// TIA Portal V19 export
FUNCTION_BLOCK "GuideLubrication_FB"   // FB155, LAD
TITLE = GUIDE LUBRICATION / MATERIAL LUBRICATION (ROLL)
// stored: Access Published, MemoryReserve 100, SetENOAutomatically false
   VAR_INPUT
      AreaInterface : "AreaInterface";
      DataIn : Struct
         PbCycleExe : Bool;
         FluxCycleDone : Bool;
         SensorLevel : Bool;
         PumpFeedbackRunning : Bool;
         PumpThermalProtection : Bool;
      END_STRUCT;
      CIn : Struct
         EnableStopInPhase : Bool;
         EnableStopProgrammed : Bool;
         MaterialCounter : LReal;
      END_STRUCT;
      Config : Struct
         EnableWngSystemOff : Bool;
         LowTankLevelDly : Time;
      END_STRUCT;
   END_VAR
   VAR_OUTPUT
      MachineInterface : "MachineInterface";
      DataOut : Struct
         M_Pump_Contactor : Bool;
         Lamp : Bool;
      END_STRUCT;
      COut : Struct
         PumpIsRunning : Bool;
      END_STRUCT;
   END_VAR
   VAR_IN_OUT
      PersistentValues : Struct
         Par : Struct
            Enable : Bool;
            CycleToExecute : Int;
            SpaceInterval : LReal;
         END_STRUCT;
      END_STRUCT;
   END_VAR
   VAR
      Sts : Struct
         AlarmsPresence : Bool;
         WarningsPresence : Bool;
         IsStandstill : Bool;
         PumpRunReq : Bool;
         LastFeed : LReal;
         PrevMatcounter : LReal;
         MaterialFed : LReal;
         PumpCnd { ExternalAccessible := 'False'; ExternalVisible := 'False'; ExternalWritable := 'False'} : Bool;
         CycleDone : Int;
      END_STRUCT;
      Ctrl : Struct
         RstAlarms : Bool;
         StopInPhase : Bool;
         StopProgrammed : Bool;
         PumpStart : Bool;
      END_STRUCT;
      Alr : Struct
         LowTankLevel : Bool;
         TimeoutCycle : Bool;
         MPump : "MotorAlr";
      END_STRUCT;
      Wng : Struct
         NoAutReady : Bool;
         SystemOff : Bool;
      END_STRUCT;
      M_Pump : "Motor";
      TON_DelayBlowerStop { S7_SetPoint := 'True'} : IEC_TIMER;
      TON_DelayPumpStop { S7_SetPoint := 'True'} : IEC_TIMER;
      TON_LowTankLevel { S7_SetPoint := 'True'} : IEC_TIMER;
      TON_CycleTimeout { S7_SetPoint := 'True'} : IEC_TIMER;
      AckRstAlarms : Bool;
      PbCycleStart_PEAux : Bool;
      CycleDone_PEAux : Bool;
   END_VAR
   VAR_TEMP
      CycleDone_PE : Bool;
   END_VAR
   VAR_TEMP   // added for the SCL form of the ladder/FBD networks
      _w1 : Bool;
   END_VAR
BEGIN

REGION Network 1 (SCL): Reset alarms command
   #Ctrl.RstAlarms := #AreaInterface.RstAlarms AND NOT #AckRstAlarms; 
   #AckRstAlarms := #AreaInterface.RstAlarms;

   IF #Ctrl.RstAlarms THEN
       #Wng.NoAutReady := FALSE;
       #Alr.LowTankLevel := FALSE;
       #Alr.TimeoutCycle := FALSE;
   END_IF;
END_REGION

REGION Network 2: Warning Pump off / Warning Pump / Blower off
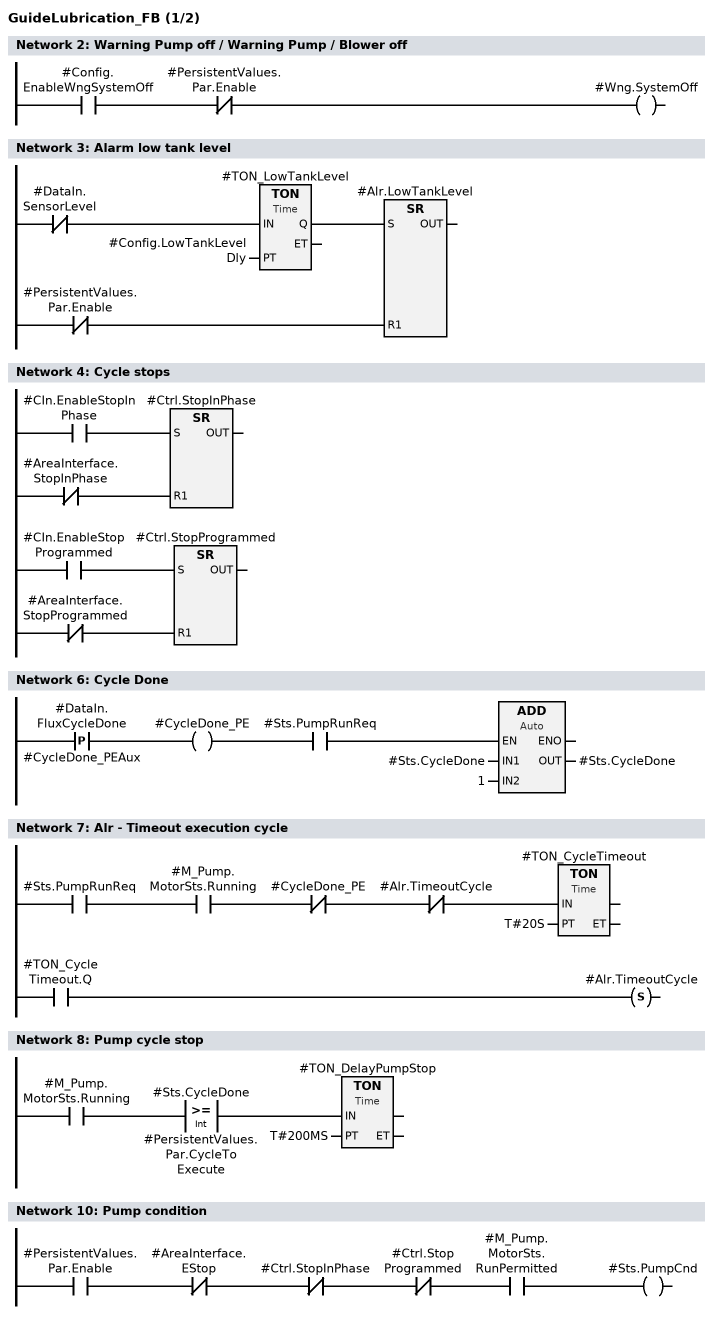
   RUNG wire#powerrail
      Contact( #Config.EnableWngSystemOff )
      I_Contact( #PersistentValues.Par.Enable )
      Coil( #Wng.SystemOff )
   END_RUNG
   // the same network as SCL:
   #Wng.SystemOff := #Config.EnableWngSystemOff AND NOT #PersistentValues.Par.Enable;
END_REGION

REGION Network 3: Alarm low tank level
   RUNG wire#powerrail
      I_Contact( #DataIn.SensorLevel )
      { S7_Templates := "time_type := Time" } #TON_LowTankLevel.TON(pt := #Config.LowTankLevelDly, et =>)
      S_SR(operand := #Alr.LowTankLevel, r1 := wire#w1)
   END_RUNG
   RUNG wire#powerrail
      I_Contact( #PersistentValues.Par.Enable )
   END_RUNG wire#w1
   // the same network as SCL:
   #TON_LowTankLevel.TON(IN := NOT #DataIn.SensorLevel, PT := #Config.LowTankLevelDly);
   IF #TON_LowTankLevel.Q THEN
       #Alr.LowTankLevel := TRUE;   // SR flip-flop
   END_IF;
   IF NOT #PersistentValues.Par.Enable THEN #Alr.LowTankLevel := FALSE; END_IF;
END_REGION

REGION Network 4: Cycle stops
   RUNG wire#powerrail
      Contact( #CIn.EnableStopInPhase )
      S_SR(operand := #Ctrl.StopInPhase, r1 := wire#w1)
   END_RUNG
   RUNG wire#powerrail
      I_Contact( #AreaInterface.StopInPhase )
   END_RUNG wire#w1
   RUNG wire#powerrail
      Contact( #CIn.EnableStopProgrammed )
      S_SR(operand := #Ctrl.StopProgrammed, r1 := wire#w2)
   END_RUNG
   RUNG wire#powerrail
      I_Contact( #AreaInterface.StopProgrammed )
   END_RUNG wire#w2
   // the same network as SCL:
   IF #CIn.EnableStopInPhase THEN
       #Ctrl.StopInPhase := TRUE;   // SR flip-flop
   END_IF;
   IF NOT #AreaInterface.StopInPhase THEN #Ctrl.StopInPhase := FALSE; END_IF;
   IF #CIn.EnableStopProgrammed THEN
       #Ctrl.StopProgrammed := TRUE;   // SR flip-flop
   END_IF;
   IF NOT #AreaInterface.StopProgrammed THEN #Ctrl.StopProgrammed := FALSE; END_IF;
END_REGION

REGION Network 5: <<< PUMP >>>
END_REGION

REGION Network 6: Cycle Done
   RUNG wire#powerrail
      P_Contact(operand := #DataIn.FluxCycleDone, bit := #CycleDone_PEAux)
      Coil( #CycleDone_PE )
      Contact( #Sts.PumpRunReq )
      Add(in1 := #Sts.CycleDone, in2 := 1, out => #Sts.CycleDone)
   END_RUNG
   // the same network as SCL:
   #_w1 := #DataIn.FluxCycleDone AND NOT #CycleDone_PEAux;   // rising edge of #DataIn.FluxCycleDone
   #CycleDone_PEAux := #DataIn.FluxCycleDone;
   #CycleDone_PE := #_w1;
   IF #_w1 AND #Sts.PumpRunReq THEN #Sts.CycleDone := #Sts.CycleDone + 1; END_IF;
END_REGION

REGION Network 7: Alr - Timeout execution cycle
   RUNG wire#powerrail
      Contact( #Sts.PumpRunReq )
      Contact( #M_Pump.MotorSts.Running )
      I_Contact( #CycleDone_PE )
      I_Contact( #Alr.TimeoutCycle )
      { S7_Templates := "time_type := Time" } #TON_CycleTimeout.TON(pt := T#20S, et =>)
   END_RUNG
   RUNG wire#powerrail
      Contact( #TON_CycleTimeout.Q )
      S_Coil( #Alr.TimeoutCycle )
   END_RUNG
   // the same network as SCL:
   #TON_CycleTimeout.TON(IN := #Sts.PumpRunReq AND #M_Pump.MotorSts.Running AND NOT #CycleDone_PE AND NOT #Alr.TimeoutCycle,
                         PT := T#20S);
   IF #TON_CycleTimeout.Q THEN #Alr.TimeoutCycle := TRUE; END_IF;
END_REGION

REGION Network 8: Pump cycle stop
   RUNG wire#powerrail
      Contact( #M_Pump.MotorSts.Running )
      { S7_Templates := "SrcType := Int" } GE_Contact(in1 := #Sts.CycleDone, in2 := #PersistentValues.Par.CycleToExecute)
      { S7_Templates := "time_type := Time" } #TON_DelayPumpStop.TON(pt := T#200MS, et =>)
   END_RUNG
   // the same network as SCL:
   #TON_DelayPumpStop.TON(IN := #M_Pump.MotorSts.Running AND (#Sts.CycleDone >= #PersistentValues.Par.CycleToExecute),
                          PT := T#200MS);
END_REGION

REGION Network 9 (SCL): Pump run request
   #Sts.LastFeed := "M_PosAMinusPosB"(PosA:=#CIn.MaterialCounter,PosB:=#Sts.PrevMatcounter,MODULE := "MATERIAL_COUNTERS_MODULE");
   #Sts.PrevMatcounter := #CIn.MaterialCounter;

   IF #Sts.LastFeed > 1000.0 THEN
       #Sts.LastFeed := 0;
   END_IF;

   #Sts.MaterialFed := #Sts.MaterialFed + #Sts.LastFeed;

   IF  #PersistentValues.Par.CycleToExecute = 0 OR #PersistentValues.Par.SpaceInterval <= 0.0 OR NOT #PersistentValues.Par.Enable THEN
       #Sts.PumpRunReq := FALSE;       
   ELSIF #TON_DelayPumpStop.Q THEN
       #Sts.PumpRunReq := FALSE;   
       #Sts.MaterialFed := 0.0;
       #Sts.CycleDone := 0;
   ELSIF NOT #Sts.PumpRunReq AND (#Sts.MaterialFed >= #PersistentValues.Par.SpaceInterval OR #DataIn.PbCycleExe) THEN
       #Sts.PumpRunReq := TRUE;
       #Sts.CycleDone := 0;
   END_IF;
END_REGION

REGION Network 10: Pump condition
   RUNG wire#powerrail
      Contact( #PersistentValues.Par.Enable )
      I_Contact( #AreaInterface.EStop )
      I_Contact( #Ctrl.StopInPhase )
      I_Contact( #Ctrl.StopProgrammed )
      Contact( #M_Pump.MotorSts.RunPermitted )
      Coil( #Sts.PumpCnd )
   END_RUNG
   // the same network as SCL:
   #Sts.PumpCnd := #PersistentValues.Par.Enable AND NOT #AreaInterface.EStop AND NOT #Ctrl.StopInPhase AND NOT #Ctrl.StopProgrammed AND #M_Pump.MotorSts.RunPermitted;
END_REGION

REGION Network 11: Pump automatic start
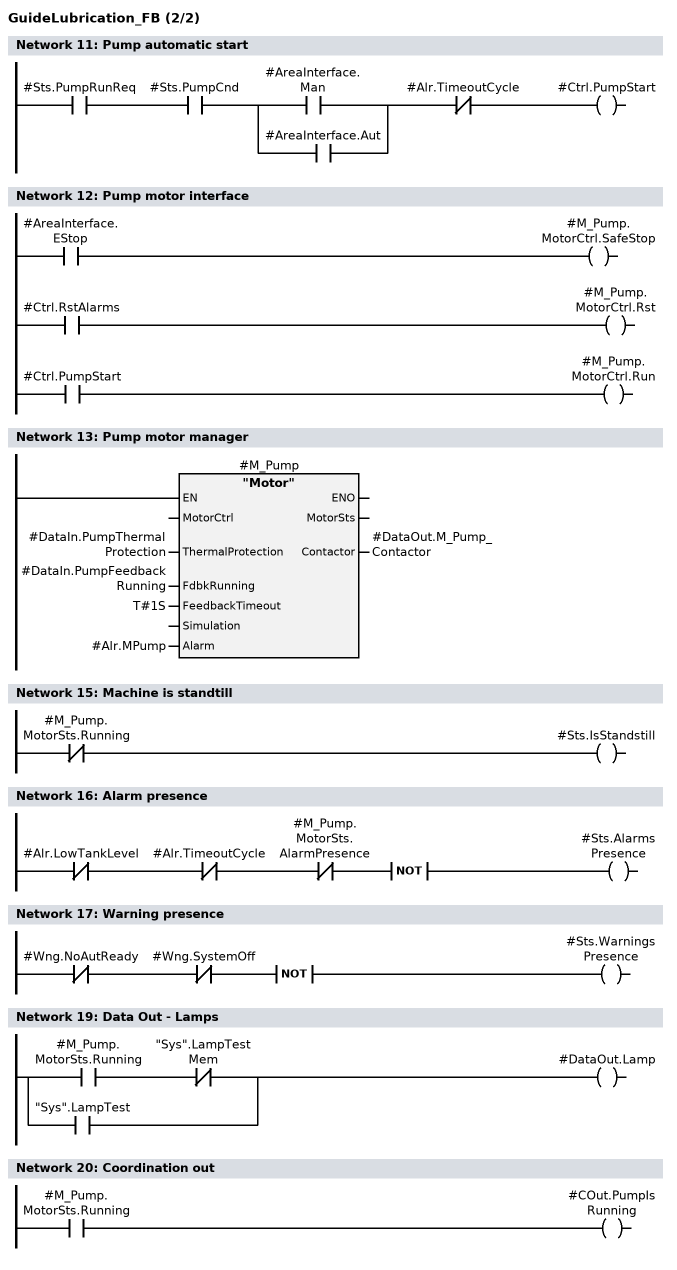
   RUNG wire#powerrail
      Contact( #Sts.PumpRunReq )
      Contact( #Sts.PumpCnd )
      wire#w1
      Contact( #AreaInterface.Man )
      wire#w2
      I_Contact( #Alr.TimeoutCycle )
      Coil( #Ctrl.PumpStart )
   END_RUNG
   RUNG wire#w1
      Contact( #AreaInterface.Aut )
   END_RUNG wire#w2
   // the same network as SCL:
   #Ctrl.PumpStart := #Sts.PumpRunReq AND #Sts.PumpCnd AND (#AreaInterface.Man OR #AreaInterface.Aut) AND NOT #Alr.TimeoutCycle;
END_REGION

REGION Network 12: Pump motor interface
   RUNG wire#powerrail
      Contact( #AreaInterface.EStop )
      Coil( #M_Pump.MotorCtrl.SafeStop )
   END_RUNG
   RUNG wire#powerrail
      Contact( #Ctrl.RstAlarms )
      Coil( #M_Pump.MotorCtrl.Rst )
   END_RUNG
   RUNG wire#powerrail
      Contact( #Ctrl.PumpStart )
      Coil( #M_Pump.MotorCtrl.Run )
   END_RUNG
   // the same network as SCL:
   #M_Pump.MotorCtrl.SafeStop := #AreaInterface.EStop;
   #M_Pump.MotorCtrl.Rst := #Ctrl.RstAlarms;
   #M_Pump.MotorCtrl.Run := #Ctrl.PumpStart;
END_REGION

REGION Network 13: Pump motor manager
   RUNG wire#powerrail
      #M_Pump(MotorCtrl :=, ThermalProtection := #DataIn.PumpThermalProtection, FdbkRunning := #DataIn.PumpFeedbackRunning, FeedbackTimeout := T#1S, Simulation :=, Alarm := #Alr.MPump, MotorSts =>, Contactor => #DataOut.M_Pump_Contactor)
   END_RUNG
   // the same network as SCL:
   #M_Pump(ThermalProtection := #DataIn.PumpThermalProtection,   // "Motor"
           FdbkRunning := #DataIn.PumpFeedbackRunning,
           FeedbackTimeout := T#1S,
           Alarm := #Alr.MPump,
           Contactor => #DataOut.M_Pump_Contactor);
END_REGION

REGION Network 14: <<< >>>
END_REGION

REGION Network 15: Machine is standtill
   RUNG wire#powerrail
      I_Contact( #M_Pump.MotorSts.Running )
      Coil( #Sts.IsStandstill )
   END_RUNG
   // the same network as SCL:
   #Sts.IsStandstill := NOT #M_Pump.MotorSts.Running;
END_REGION

REGION Network 16: Alarm presence
   RUNG wire#powerrail
      I_Contact( #Alr.LowTankLevel )
      I_Contact( #Alr.TimeoutCycle )
      I_Contact( #M_Pump.MotorSts.AlarmPresence )
      Not()
      Coil( #Sts.AlarmsPresence )
   END_RUNG
   // the same network as SCL:
   #Sts.AlarmsPresence := NOT (NOT #Alr.LowTankLevel AND NOT #Alr.TimeoutCycle AND NOT #M_Pump.MotorSts.AlarmPresence);
END_REGION

REGION Network 17: Warning presence
   RUNG wire#powerrail
      I_Contact( #Wng.NoAutReady )
      I_Contact( #Wng.SystemOff )
      Not()
      Coil( #Sts.WarningsPresence )
   END_RUNG
   // the same network as SCL:
   #Sts.WarningsPresence := NOT (NOT #Wng.NoAutReady AND NOT #Wng.SystemOff);
END_REGION

REGION Network 18 (SCL): Collect machine to area interface
   // Status machine ready
   #MachineInterface.AutReady := #AreaInterface.Aut AND NOT #Sts.AlarmsPresence;
   // Status machine aborting
   #MachineInterface.Aborting := #Sts.AlarmsPresence;
   // Status Ack Stop in phase
   #MachineInterface.AckStopInPhase := #Ctrl.StopInPhase AND #MachineInterface.MotionsStandStill;
   // Status Ack Stop programmed
   #MachineInterface.AckStopProgrammed := #Ctrl.StopProgrammed AND #MachineInterface.MotionsStandStill;
   // Status Motion standtill
   #MachineInterface.MotionsStandStill := #Sts.IsStandstill;
   // Status Alarm presence
   #MachineInterface.AlarmsPresence := #Sts.AlarmsPresence;
   // Status Warning presence
   #MachineInterface.WarningPresence := #Sts.WarningsPresence;

   // Warning machine not automatic ready
   IF #AreaInterface.CheckAutReady AND NOT #MachineInterface.AutReady THEN
     #Wng.NoAutReady := false;
   END_IF;
END_REGION

REGION Network 19: Data Out - Lamps
   RUNG wire#powerrail
      Contact( #M_Pump.MotorSts.Running )
      I_Contact( "Sys".LampTestMem )
      wire#w1
      Coil( #DataOut.Lamp )
   END_RUNG
   RUNG wire#powerrail
      Contact( "Sys".LampTest )
   END_RUNG wire#w1
   // the same network as SCL:
   #DataOut.Lamp := (#M_Pump.MotorSts.Running AND NOT "Sys".LampTestMem) OR "Sys".LampTest;
END_REGION

REGION Network 20: Coordination out
   RUNG wire#powerrail
      Contact( #M_Pump.MotorSts.Running )
      Coil( #COut.PumpIsRunning )
   END_RUNG
   // the same network as SCL:
   #COut.PumpIsRunning := #M_Pump.MotorSts.Running;
END_REGION
END_FUNCTION_BLOCK
